TYPE HMI_WRN_RbtFanucUnloading EXTENDS HMI_WRN_RbtFanuc:
STRUCT
	;//add custom bools on top of library block here
END_STRUCT
END_TYPE

(* stored: Version 1.1.0.1
   DUT HMI_WRN_RbtFanucUnloading: Id {c5f18d46-4cbb-45d7-b0b7-892b3d806064} *)
